// TwinCAT 3 PLC project Lab1
// ProgramVersion: 3.1.4023.0
// libraries:
//   Tc2_Standard, * (Beckhoff Automation GmbH)
//   Tc2_System, * (Beckhoff Automation GmbH)
//   Tc3_Module, * (Beckhoff Automation GmbH)
//   VisuDialogs, * (System)
// project tree:
//   / GlobalTextList.TcGTLO, PlcTask.TcTTO (not stored), Visualization Manager.TcVMO (not stored)
//   GVLs/ Inputs.TcGVL, Outputs.TcGVL, Parameters.TcGVL
//   POUs/ CraneSimulation.TcPOU, MAIN.TcPOU
//   VISUs/ CraneHMI.TcVIS
// real-time tasks:
//   TASK PlcTask: cycle T#10ms, priority 20, ADS port 350

// ---- GVLs/Inputs.TcGVL
{attribute 'qualified_only'}
VAR_GLOBAL
	bEnableSimulation : BOOL; 
	bStartSimulation : BOOL; 
	fCylinderVelocityReference : LREAL; 
END_VAR

// ---- GVLs/Outputs.TcGVL
{attribute 'qualified_only'}
VAR_GLOBAL
	fSimulationTime : LREAL; 
	bSimulationRunning : BOOL;
	fCylinderVelocity : LREAL;
	fCylinderPosition : LREAL;
	pt0_x : INT;
	pt0_y : INT;
	pt1_x : INT;
	pt1_y : INT; 
END_VAR

// ---- GVLs/Parameters.TcGVL
{attribute 'qualified_only'}
VAR_GLOBAL
	fCyclicTime : LREAL := 0.01; 
	fPistonScale : LREAL;
END_VAR

// ---- POUs/CraneSimulation.TcPOU
PROGRAM CraneSimulation
VAR
	fTime : LREAL; 	
	bRunning : BOOL;
	fPosition : LREAL; 
	fInitialPosition : LREAL; 
	fInitialVelocity : LREAL; 
END_VAR

IF Inputs.bStartSimulation THEN
	fTime := fTime + Parameters.fCyclicTime;
ELSE
	fTime := 0; 	
END_IF

IF fTime > 0 THEN 
	bRunning := TRUE;
ELSE
	bRunning := FALSE;
END_IF

fPosition := Inputs.fCylinderVelocityReference * (fTime * fTime)/2 + fInitialVelocity * fTime + fInitialPosition;

IF fPosition >= 1 THEN
	Outputs.fCylinderPosition := 1;	
ELSIF fPosition <= 0 THEN
	Outputs.fCylinderPosition := 0; 
ELSE	
	Outputs.fCylinderPosition := fPosition;
END_IF

Outputs.bSimulationRunning := bRunning;  
Outputs.fSimulationTime := fTime; 
Outputs.fCylinderVelocity := Inputs.fCylinderVelocityReference;
Outputs.pt1_y := LREAL_TO_INT(Outputs.fCylinderPosition * Parameters.fPistonScale);

END_PROGRAM

// ---- POUs/MAIN.TcPOU
PROGRAM MAIN
VAR
END_VAR

IF Inputs.bEnable THEN
	CraneCommander();
END_IF

END_PROGRAM

// ---- GlobalTextList.TcGTLO
TEXTLIST GlobalTextList
  624 = '%0.1f'
  198 = '%f'
  949 = '%i'
  819 = '%s'
  236 = 'Clock: %s [s]'
  752 = 'Cylinder Velocity Reference: %0.0001f [m/s]'
  954 = 'Cylinder Velocity Reference: %0.01f [m/s]'
  105 = 'Cylinder Velocity Reference: %0.1f [m/s]'
  755 = 'Cylinder Velocity Reference: %0.1s [m/s]'
  25 = 'Cylinder Velocity Reference: %f [m/s]'
  30 = 'Cylinder Velocity Reference: %i'
  903 = 'Cylinder Velocity Reference: %s'
  128 = 'Cylinder Velocity Reference: %s [m/s]'
  353 = 'Enable'
  409 = 'ENABLE'
  310 = 'RUNNING'
  466 = 'Simulation'
  279 = 'Start'
  868 = 'START'
  978 = 'Started'
  495 = 'Time: %0.1f [s]'
  221 = 'Time: %f [s]'
  61 = 'Time: %i [s]'
  725 = 'Time: %s [s]'
END_TEXTLIST

// ---- VISUs/CraneHMI.TcVIS
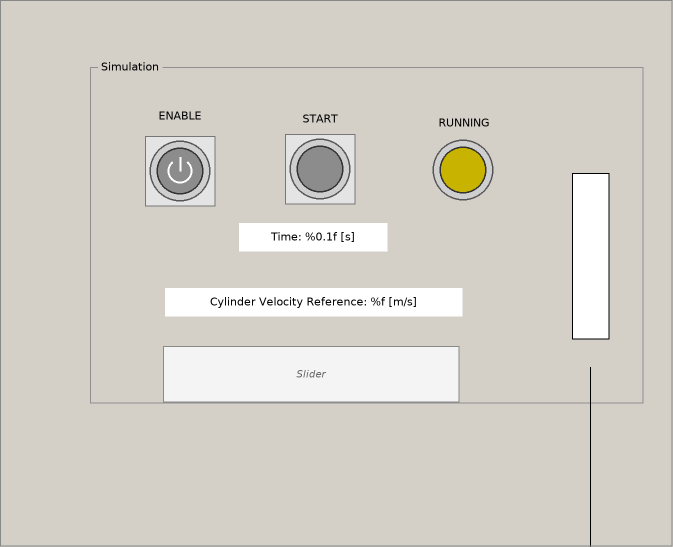
VISUALIZATION CraneHMI  // 673x547
    Rectangle (507,238 166x37), angle 270
        p2738717112: Outputs.fCylinderPosition
    GroupBox (90,59 553x344), "Simulation"
        PowerSwitch (55,77 70x70), variable: Inputs.bEnableSimulation, behaviour: TOGGLE, style: Switch-PowerSwitch-Gray
        PushSwitch (195,75 70x70), variable: Inputs.bStartSimulation, behaviour: TOGGLE, style: Switch-PushSwitch-Gray
        Lamp1 (338,76 70x70), variable: Outputs.bSimulationRunning, style: Lamp-Lamp1-Yellow
        Textfield (74,228 299x30), "Cylinder Velocity Reference: %f [m/s]", text variable: Inputs.fCylinderVelocityReference
            OnMouseClick: write the text variable via Default
        Label (15,42 150x30), "ENABLE"
        Label (155,45 150x30), "START"
        Label (299,49 150x30), "RUNNING"
        Textfield (148,163 150x30), "Time: %0.1f [s]", text variable: Outputs.fSimulationTime
        Slider (73,287 296x56), variable: Inputs.fCylinderVelocityReference, scale -0.1..0.1
    Line (590,367) (590,547)
        p1126004900: Outputs.pt1_y
        p3528305787: Outputs.pt0_x
        p2773130477: Outputs.pt0_y
        p874137650: Outputs.pt1_x
END_VISUALIZATION
